FUNCTION_BLOCK PUBLIC FB_CraneModeControlBox IMPLEMENTS I_Mode
VAR_INPUT
END_VAR
VAR_OUTPUT
END_VAR
VAR
END_VAR

{warning 'add method implementation '}
METHOD Auto
VAR_INPUT
	bAuto : BOOL := 0;
END_VAR
END_METHOD

{warning 'add method implementation '}
METHOD Manual
VAR_INPUT
	bManual : BOOL := 0;
END_VAR
END_METHOD

{warning 'add method implementation '}
METHOD Off
VAR_INPUT
	bOff : BOOL := 1;
END_VAR
END_METHOD

END_FUNCTION_BLOCK

(* stored: Version 1.1.0.1, ProductVersion 3.1.4024.9
   POU FB_CraneModeControlBox: Id {002e0df9-916a-46f2-98e4-26176fe232e3}, SpecialFunc None
   Method Auto: Id {aec474cc-52a2-4075-807a-92a54a3c6393}
   Method Manual: Id {c68168bd-1e76-4dfe-a72c-92fb65666c3e}
   Method Off: Id {15e5efa7-2ccb-482e-bd29-a66b5f0bc569} *)
